// TIA Portal V19 export
TYPE "LEXCHANGETRAY_typeSr1000ProfinetTelegram_parameterBankNumber"
// stored: Access Published
   STRUCT
      parameterBytes : Array[0..1] of Byte;
   END_STRUCT;
END_TYPE
